FUNCTION_BLOCK Test_TStreamAdd_Read_ULINT EXTENDS TUnitTestBase
VAR
    Stream : TStream(StreamLength := 2);
END_VAR



Stream.Init(2);

Stream.Add_ULINT(123456789);
    
Assertion.AssertEquals_UDINT(
    Expected := 8,
    Actual := Stream.Position,
    VariableName := 'Stream.Position');
    
Stream.Seek(0);

Assertion.AssertEquals_ULINT(
    Expected := 123456789,
    Actual := Stream.Read_ULINT(),
    VariableName := 'Stream.Read_ULINT()');
    
Assertion.AssertEquals_UDINT(
    Expected := 8,
    Actual := Stream.Position,
    VariableName := 'Stream.Position');
    
    
TestFinished();

END_FUNCTION_BLOCK

(* stored: Version 1.1.0.1, ProductVersion 3.1.4024.4
   POU Test_TStreamAdd_Read_ULINT: Id {b446ba35-af1a-476f-a38c-a057c6d4ef61}, SpecialFunc None *)
